FUNCTION_BLOCK GasBurner
  (* Standard: 61499-2 *)
  (* Version 0.1, 2015-00-10, syy, syy-PC *)
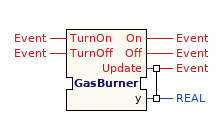
  EVENT_INPUT
    TurnOn;
    TurnOff;
  END_EVENT
  EVENT_OUTPUT
    On;
    Off;
    Update WITH y;
  END_EVENT
  VAR_OUTPUT
    y : REAL;
  END_VAR
  VAR
    d : REAL;
  END_VAR
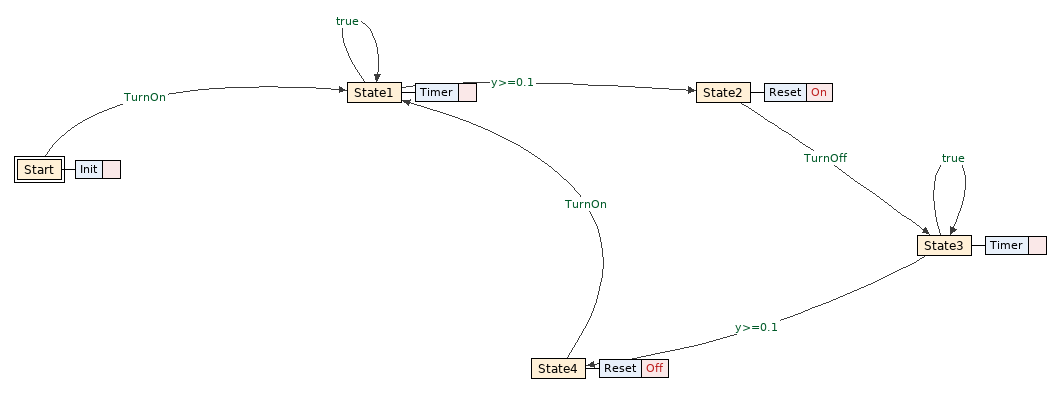
  EC_STATES
    Start : Init;
    State1 : Timer;
    State2 : Reset -> On;
    State3 : Timer;
    State4 : Reset -> Off;
  END_STATES
  EC_TRANSITIONS
    Start TO State1 := TurnOn;
    State1 TO State2 := y>=0.1;
    State1 TO State1 := true;
    State2 TO State3 := TurnOff;
    State3 TO State4 := y>=0.1;
    State3 TO State3 := true;
    State4 TO State1 := TurnOn;
  END_TRANSITIONS
  ALGORITHM Init IN C:
me->y=0;
me->d=0.01;
  END_ALGORITHM
  ALGORITHM Timer IN C:
me->y=(float) me->y+me->d;
//printf("timer : %f\n", me->y);
  END_ALGORITHM
  ALGORITHM Reset IN C:
//printf("signal transfered\n");
me->y=0;
  END_ALGORITHM
END_FUNCTION_BLOCK
